% RSLogix 500 project P1.RSS, saved by version 8.30.00.16 %
PROJECT "P1"    % processor: Bul.1763 MicroLogix 1100 Series B %

PROGRAM FILES
  LAD 2   3 rungs
  LAD 3 "IO"  5 rungs
  LAD 4 "CTRL"  11 rungs

DATA FILES
  O0 OUTPUT  4 elements
  I1 INPUT  6 elements
  S2 STATUS  66 elements
  B3 BINARY  1 elements
  T4 TIMER  4 elements
  C5 COUNTER  1 elements
  R6 CONTROL  1 elements
  N7 INTEGER  1 elements
  F8 FLOAT  1 elements

LADDER 2
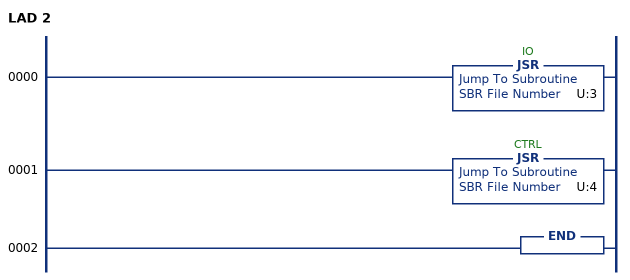
% Rung: 0 %
SOR JSR U:3 EOR
%   U:3  "IO" %
% Rung: 1 %
SOR JSR U:4 EOR
%   U:4  "CTRL" %
% Rung: 2 %
SOR END EOR

LADDER 3 "IO"
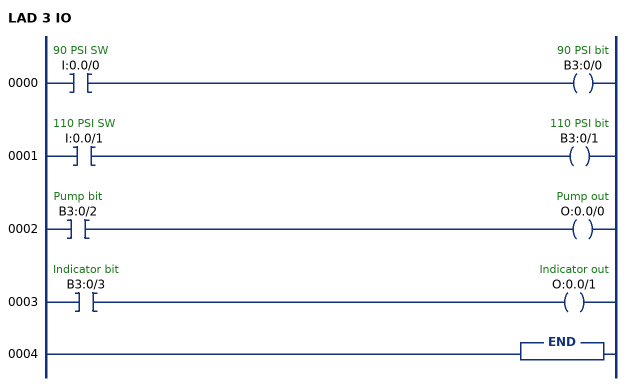
% Rung: 0 %
SOR XIC I:0.0/0 OTE B3:0/0 EOR
%   I:0.0/0  "90 PSI SW" %
%   B3:0/0  "90 PSI bit" %
% Rung: 1 %
SOR XIC I:0.0/1 OTE B3:0/1 EOR
%   I:0.0/1  "110 PSI SW" %
%   B3:0/1  "110 PSI bit" %
% Rung: 2 %
SOR XIC B3:0/2 OTE O:0.0/0 EOR
%   B3:0/2  "Pump bit" %
%   O:0.0/0  "Pump out" %
% Rung: 3 %
SOR XIC B3:0/3 OTE O:0.0/1 EOR
%   B3:0/3  "Indicator bit" %
%   O:0.0/1  "Indicator out" %
% Rung: 4 %
SOR END EOR

LADDER 4 "CTRL"
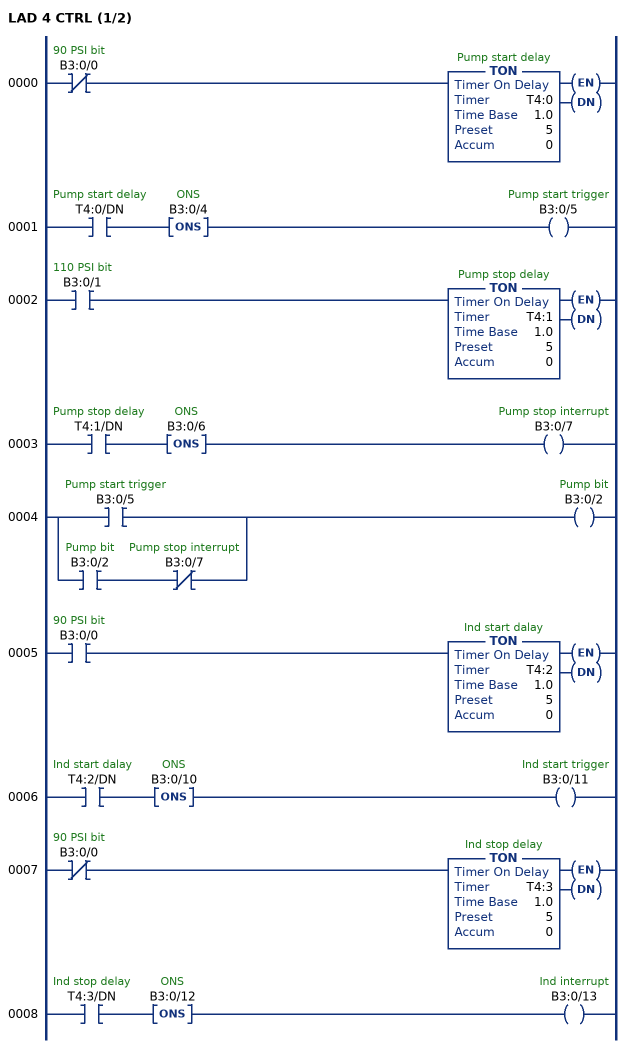
% Rung: 0 %
SOR XIO B3:0/0 TON T4:0 1.0 5 0 EOR
%   B3:0/0  "90 PSI bit" %
%   T4:0  "Pump start delay" %
% Rung: 1 %
SOR XIC T4:0/DN ONS B3:0/4 OTE B3:0/5 EOR
%   T4:0  "Pump start delay" %
%   B3:0/4  "ONS" %
%   B3:0/5  "Pump start trigger" %
% Rung: 2 %
SOR XIC B3:0/1 TON T4:1 1.0 5 0 EOR
%   B3:0/1  "110 PSI bit" %
%   T4:1  "Pump stop delay" %
% Rung: 3 %
SOR XIC T4:1/DN ONS B3:0/6 OTE B3:0/7 EOR
%   T4:1  "Pump stop delay" %
%   B3:0/6  "ONS" %
%   B3:0/7  "Pump stop interrupt" %
% Rung: 4 %
SOR BST XIC B3:0/5 NXB XIC B3:0/2 XIO B3:0/7 BND OTE B3:0/2 EOR
%   B3:0/5  "Pump start trigger" %
%   B3:0/2  "Pump bit" %
%   B3:0/7  "Pump stop interrupt" %
% Rung: 5 %
SOR XIC B3:0/0 TON T4:2 1.0 5 0 EOR
%   B3:0/0  "90 PSI bit" %
%   T4:2  "Ind start dalay" %
% Rung: 6 %
SOR XIC T4:2/DN ONS B3:0/10 OTE B3:0/11 EOR
%   T4:2  "Ind start dalay" %
%   B3:0/10  "ONS" %
%   B3:0/11  "Ind start trigger" %
% Rung: 7 %
SOR XIO B3:0/0 TON T4:3 1.0 5 0 EOR
%   B3:0/0  "90 PSI bit" %
%   T4:3  "Ind stop delay" %
% Rung: 8 %
SOR XIC T4:3/DN ONS B3:0/12 OTE B3:0/13 EOR
%   T4:3  "Ind stop delay" %
%   B3:0/12  "ONS" %
%   B3:0/13  "Ind interrupt" %

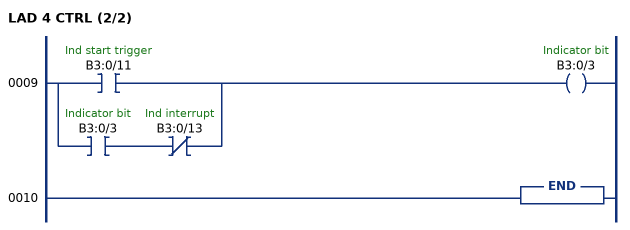
% Rung: 9 %
SOR BST XIC B3:0/11 NXB XIC B3:0/3 XIO B3:0/13 BND OTE B3:0/3 EOR
%   B3:0/11  "Ind start trigger" %
%   B3:0/3  "Indicator bit" %
%   B3:0/13  "Ind interrupt" %
% Rung: 10 %
SOR END EOR

OTHER DOCUMENTED ADDRESSES
  B3:0/8  "ONS"
  B3:0/9  "Ind start trigger"

DATA TABLE (non-zero values as saved)
DATA T4
% .PRE .ACC %
% T4:0 % 5 0
% T4:1 % 5 0
% T4:2 % 5 0
% T4:3 % 5 0
